// TIA Portal project "Clasificadora_Peso" (V16)

(* hardware
DEVICE "S71500/ET200MP station_1"  S7-1500 station
   slot 0: "Perfil soporte_0"  Rack  6ES7 590-1***0-0AA0
   slot 1: "PLC_Clasificadora_Peso"  CPU 1511-1 PN  6ES7 511-1AK02-0AB0  V2.5
      slot 3: "Display de la CPU_1"  6ES7591-1AA00-0AA0
      slot 32768: "Interfaz PROFINET_1"  X1
         slot 32769: "Puerto_1"  X1 P1
         slot 32770: "Puerto_2"  X1 P2
*)

// ===== PLC "PLC_Clasificadora_Peso"  CPU 1511-1 PN =====

VAR_GLOBAL   // PLC tag table "Tabla de variables estándar"
   "Cinta_Entrada_1" AT %Q0.1 : Bool;
   "Cinta_Entrada_2" AT %Q0.2 : Bool;
   "Piston_1" AT %Q0.3 : Bool;
   "Piston_2" AT %Q0.4 : Bool;
   "Cinta_Peso_1" AT %Q0.5 : Bool;
   "Cinta_Peso_2" AT %Q0.6 : Bool;
   "Cinta_Salida_1" AT %Q0.7 : Bool;
   "Cinta_Salida_2" AT %Q1.0 : Bool;
   "Start_HMI" AT %M0.1 : Bool;
   "Stop_HMI" AT %M0.2 : Bool;
   "Emitter_1" AT %Q1.1 : Bool;
   "Emitter_2" AT %Q1.2 : Bool;
   "Peso" AT %IW100 : Word;
   "Peso_Normal" AT %ID100 : Real;
   "Peso_Entero" AT %MW102 : Word;
   "Sensor_Clasificador" AT %I0.3 : Bool;
   "Pieza_1" AT %M0.3 : Bool;
   "Pieza_2" AT %M0.4 : Bool;
   "Piston_Extendido" AT %I0.4 : Bool;
   "Sensor_Peso" AT %I0.5 : Bool;
   "Piston_Retraido" AT %I0.6 : Bool;
   "Sensor_Salida" AT %I0.7 : Bool;
   "Peso_Real" AT %MD104 : Real;
   "Start" AT %I1.0 : Bool;
   "Stop" AT %I1.1 : Bool;
   "Start_light" AT %Q1.3 : Bool;
   "Stop_light" AT %Q1.4 : Bool;
END_VAR

ORGANIZATION_BLOCK "Main"   // OB1, LAD, ProgramCycle
TITLE = "Main Program Sweep (Cycle)"
{ S7_Optimized_Access := 'TRUE' }
VERSION : 0.1
   VAR_INPUT
      Initial_Call : Bool;   // Initial call of this OB
      Remanence : Bool;   // =True, if remanent data are available
   END_VAR
   VAR_TEMP   // added for the SCL form of the ladder/FBD networks
      _w1 : Bool;
   END_VAR
BEGIN

REGION Network 1
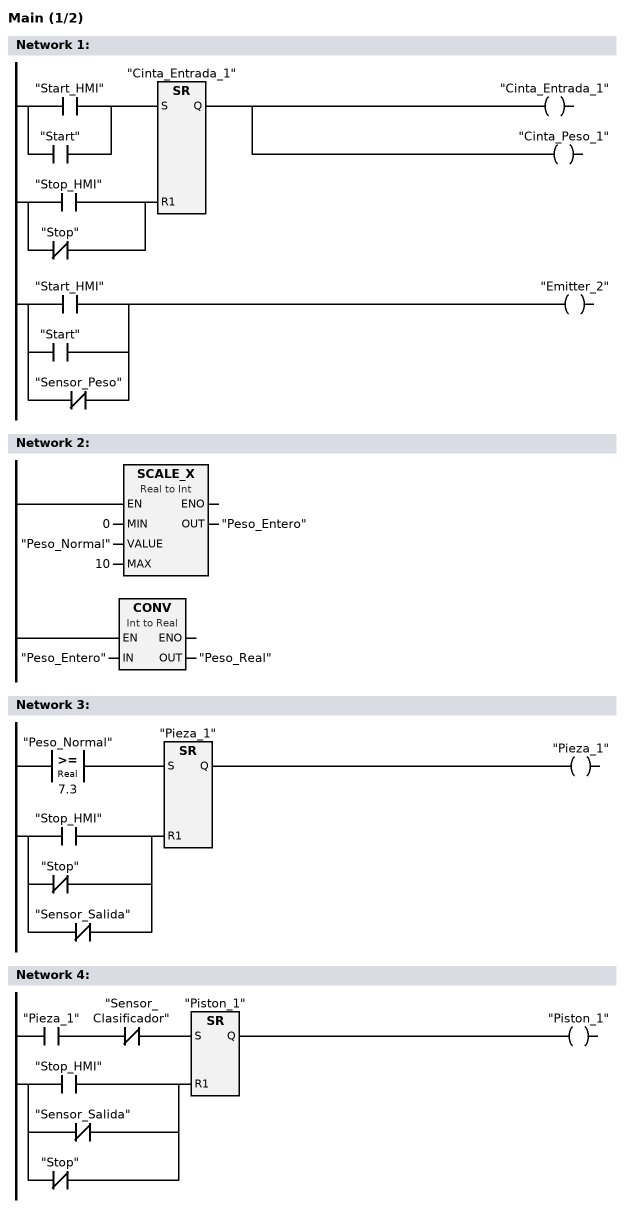
   RUNG wire#powerrail
      Contact( "Start_HMI" )
      wire#w1
      S_SR(operand := "Cinta_Entrada_1", r1 := wire#w2)
      wire#w3
      Coil( "Cinta_Entrada_1" )
   END_RUNG
   RUNG wire#powerrail
      Contact( "Start" )
   END_RUNG wire#w1
   RUNG wire#powerrail
      Contact( "Stop_HMI" )
   END_RUNG wire#w2
   RUNG wire#powerrail
      I_Contact( "Stop" )
   END_RUNG wire#w2
   RUNG wire#w3
      Coil( "Cinta_Peso_1" )
   END_RUNG
   RUNG wire#powerrail
      Contact( "Start_HMI" )
      wire#w4
      Coil( "Emitter_2" )
   END_RUNG
   RUNG wire#powerrail
      Contact( "Start" )
   END_RUNG wire#w4
   RUNG wire#powerrail
      I_Contact( "Sensor_Peso" )
   END_RUNG wire#w4
   // the same network as SCL:
   IF "Start_HMI" OR "Start" THEN
       "Cinta_Entrada_1" := TRUE;   // SR flip-flop
   END_IF;
   IF "Stop_HMI" OR NOT "Stop" THEN "Cinta_Entrada_1" := FALSE; END_IF;
   #_w1 := "Cinta_Entrada_1";
   "Cinta_Entrada_1" := "Cinta_Entrada_1";
   "Cinta_Peso_1" := #_w1;
   "Emitter_2" := "Start_HMI" OR "Start" OR NOT "Sensor_Peso";
END_REGION

REGION Network 2
   RUNG wire#powerrail
      { S7_Templates := "[SrcType := Real, DestType := Int]" } Scale(min := 0, value := "Peso_Normal", max := 10, out => "Peso_Entero")
   END_RUNG
   RUNG wire#powerrail
      { S7_Templates := "[SrcType := Int, DestType := Real]" } Convert(in := "Peso_Entero", out => "Peso_Real")
   END_RUNG
   // the same network as SCL:
   "Peso_Entero" := SCALE_X(MIN := 0, VALUE := "Peso_Normal", MAX := 10);
   "Peso_Real" := INT_TO_REAL("Peso_Entero");
END_REGION

REGION Network 3
   RUNG wire#powerrail
      { S7_Templates := "SrcType := Real" } GE_Contact(in1 := "Peso_Normal", in2 := 7.3)
      S_SR(operand := "Pieza_1", r1 := wire#w1)
      Coil( "Pieza_1" )
   END_RUNG
   RUNG wire#powerrail
      Contact( "Stop_HMI" )
   END_RUNG wire#w1
   RUNG wire#powerrail
      I_Contact( "Stop" )
   END_RUNG wire#w1
   RUNG wire#powerrail
      I_Contact( "Sensor_Salida" )
   END_RUNG wire#w1
   // the same network as SCL:
   IF "Peso_Normal" >= 7.3 THEN
       "Pieza_1" := TRUE;   // SR flip-flop
   END_IF;
   IF "Stop_HMI" OR NOT "Stop" OR NOT "Sensor_Salida" THEN "Pieza_1" := FALSE; END_IF;
   "Pieza_1" := "Pieza_1";
END_REGION

REGION Network 4
   RUNG wire#powerrail
      Contact( "Pieza_1" )
      I_Contact( "Sensor_Clasificador" )
      S_SR(operand := "Piston_1", r1 := wire#w1)
      Coil( "Piston_1" )
   END_RUNG
   RUNG wire#powerrail
      Contact( "Stop_HMI" )
   END_RUNG wire#w1
   RUNG wire#powerrail
      I_Contact( "Sensor_Salida" )
   END_RUNG wire#w1
   RUNG wire#powerrail
      I_Contact( "Stop" )
   END_RUNG wire#w1
   // the same network as SCL:
   IF "Pieza_1" AND NOT "Sensor_Clasificador" THEN
       "Piston_1" := TRUE;   // SR flip-flop
   END_IF;
   IF "Stop_HMI" OR NOT "Sensor_Salida" OR NOT "Stop" THEN "Piston_1" := FALSE; END_IF;
   "Piston_1" := "Piston_1";
END_REGION

REGION Network 5
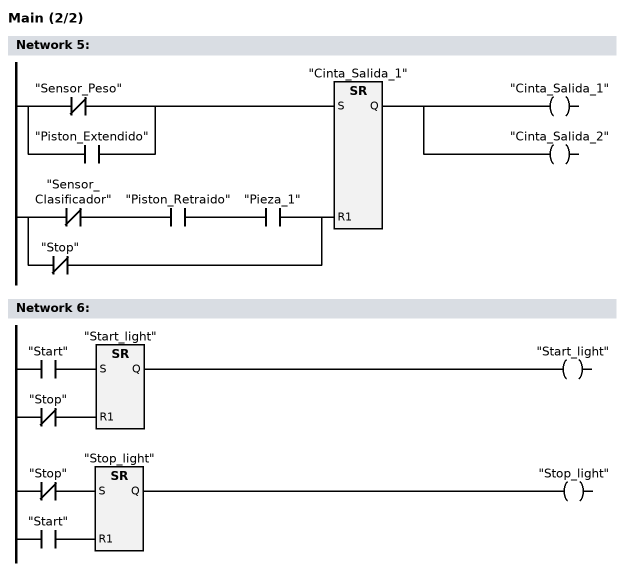
   RUNG wire#powerrail
      I_Contact( "Sensor_Peso" )
      wire#w1
      S_SR(operand := "Cinta_Salida_1", r1 := wire#w2)
      wire#w3
      Coil( "Cinta_Salida_1" )
   END_RUNG
   RUNG wire#powerrail
      Contact( "Piston_Extendido" )
   END_RUNG wire#w1
   RUNG wire#powerrail
      I_Contact( "Sensor_Clasificador" )
      Contact( "Piston_Retraido" )
      Contact( "Pieza_1" )
   END_RUNG wire#w2
   RUNG wire#powerrail
      I_Contact( "Stop" )
   END_RUNG wire#w2
   RUNG wire#w3
      Coil( "Cinta_Salida_2" )
   END_RUNG
   // the same network as SCL:
   IF NOT "Sensor_Peso" OR "Piston_Extendido" THEN
       "Cinta_Salida_1" := TRUE;   // SR flip-flop
   END_IF;
   IF (NOT "Sensor_Clasificador" AND "Piston_Retraido" AND "Pieza_1") OR NOT "Stop" THEN
       "Cinta_Salida_1" := FALSE;
   END_IF;
   #_w1 := "Cinta_Salida_1";
   "Cinta_Salida_1" := "Cinta_Salida_1";
   "Cinta_Salida_2" := #_w1;
END_REGION

REGION Network 6
   RUNG wire#powerrail
      Contact( "Start" )
      S_SR(operand := "Start_light", r1 := wire#w1)
      Coil( "Start_light" )
   END_RUNG
   RUNG wire#powerrail
      I_Contact( "Stop" )
   END_RUNG wire#w1
   RUNG wire#powerrail
      I_Contact( "Stop" )
      S_SR(operand := "Stop_light", r1 := wire#w2)
      Coil( "Stop_light" )
   END_RUNG
   RUNG wire#powerrail
      Contact( "Start" )
   END_RUNG wire#w2
   // the same network as SCL:
   IF "Start" THEN
       "Start_light" := TRUE;   // SR flip-flop
   END_IF;
   IF NOT "Stop" THEN "Start_light" := FALSE; END_IF;
   "Start_light" := "Start_light";
   IF NOT "Stop" THEN
       "Stop_light" := TRUE;   // SR flip-flop
   END_IF;
   IF "Start" THEN "Stop_light" := FALSE; END_IF;
   "Stop_light" := "Stop_light";
END_REGION
END_ORGANIZATION_BLOCK